// TIA Portal V16 export
// export: Created 2024-09-05T17:39:08.4825116Z, ExportSetting WithDefaults, DisplayName Totally Integrated Automation Portal, DisplayVersion V16 Update 6, DisplayName TIA Portal Version Control Interface, DisplayVersion V16 Update 2, DisplayName TIA Portal Openness, DisplayVersion V16 Update 6, DisplayName STEP 7 Professional, DisplayVersion V16 Update 6, DisplayName STEP 7 Safety, DisplayVersion V16, DisplayName WinCC Advanced, DisplayVersion V16 Update 6
DATA_BLOCK "PartHolderData"   // DB21
{ S7_Optimized_Access := 'TRUE' }
VERSION : 0.1
// stored: AutoNumber true, DBAccessibleFromOPCUA true, IsOnlyStoredInLoadMemory false, IsRetainMemResEnabled false, IsWriteProtectedInAS false, MemoryReserve 100
   VAR RETAIN
      OkUpperStockAmountSideA : USInt := 1;
      OkLowerStockAmountSideA : USInt := 0;
      NOKBoxAmount : USInt := 1;
   END_VAR
   VAR
      NOKBoxFull : Bool := FALSE;
      ConfirmEmptyOKStock : Bool := FALSE;
      ConfirmEmptyNOKBox : Bool := FALSE;
      EmptyOKStockConfirmed : Bool := FALSE;
      EmptyNOKBoxConfirmed : Bool := FALSE;
      NOKBoxActivated : Bool := FALSE;
      NOKBoxPesent : Bool := TRUE;
      OKholderPresent : Bool := TRUE;
      OKholderReadySideA : Bool := FALSE;
      OKholderReadySideB : Bool;
   END_VAR
   VAR RETAIN
      OkUpperStockAmountSideB : USInt := 0;
      OkLowerStockAmountSideB : USInt := 0;
   END_VAR
BEGIN
END_DATA_BLOCK
